TYPE Union_UDINT :
UNION
	value : UDINT ;
	packed : ARRAY[0..3] OF BYTE;
END_UNION
END_TYPE

(* stored: Version 1.1.0.1, ProductVersion 3.1.4024.13
   DUT Union_UDINT: Id {84233d4d-eccb-428f-9af3-961a06e07a2a} *)
